{attribute 'GeneratedUsingTerminal: EL6201-0000-0017'}
{attribute addProperty BoxType "EL6201-0000-0017"}
{attribute addProperty Id "Slave_6A_DO0BOOL1Slave_6A_DO1BOOL1Slave_6A_DO2BOOL1Slave_6A_DO3BOOL1Slave_6B_DO0BOOL1Slave_6B_DO1BOOL1Slave_6B_DO2BOOL1Slave_6B_DO3BOOL1"}
{attribute addProperty CRC "2158889732"}
{attribute addProperty Size "8"}
TYPE Slave_6_Outputs_80AE0B04 :
STRUCT
	{attribute addProperty Name "Slave_6A_DO0"}
	Slave_6A_DO0 : BOOL;
	{attribute addProperty Name "Slave_6A_DO1"}
	Slave_6A_DO1 : BOOL;
	{attribute addProperty Name "Slave_6A_DO2"}
	Slave_6A_DO2 : BOOL;
	{attribute addProperty Name "Slave_6A_DO3"}
	Slave_6A_DO3 : BOOL;
	{attribute addProperty Name "Slave_6B_DO0"}
	Slave_6B_DO0 : BOOL;
	{attribute addProperty Name "Slave_6B_DO1"}
	Slave_6B_DO1 : BOOL;
	{attribute addProperty Name "Slave_6B_DO2"}
	Slave_6B_DO2 : BOOL;
	{attribute addProperty Name "Slave_6B_DO3"}
	Slave_6B_DO3 : BOOL;
END_STRUCT
END_TYPE

(* stored: Version 1.2.0.0, ProductVersion 3.1.4024.9
   DUT Slave_6_Outputs_80AE0B04: Id {1e909065-577d-4c01-b9de-767b81817af8} *)
